# EPICS autosave request: iocBoot/ioc13DDIA30/auto_positions.req
file "CARS_motor_positions.req",         P=$(P), M=m1
file "CARS_motor_positions.req",         P=$(P), M=m2
